FUNCTION_BLOCK Template
  (* Version 1.0, 2005-04-08, Author Name, Chalmers *)
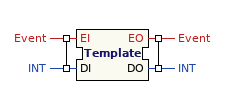
  EVENT_INPUT
    EI WITH DI;
  END_EVENT
  EVENT_OUTPUT
    EO WITH DO;
  END_EVENT
  VAR_INPUT
    DI : INT;
  END_VAR
  VAR_OUTPUT
    DO : INT;
  END_VAR
  VAR
    invoked : INT;
  END_VAR
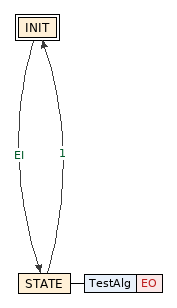
  EC_STATES
    INIT;
    STATE : TestAlg -> EO;
  END_STATES
  EC_TRANSITIONS
    INIT TO STATE := EI;
    STATE TO INIT := 1;
  END_TRANSITIONS
  ALGORITHM TestAlg IN Java:
        invoked = invoked + 1;
		DO = DI + 1;
		System.out.println("TestType.fbt:TestAlg;invoked: " + invoked + " times.");
		System.out.println("TestType.fbt:TestAlg; DO:" + DO + ".");
  END_ALGORITHM
END_FUNCTION_BLOCK
